// TIA Portal V18 export
// export: Created 2026-06-08T16:32:19.8720491Z, ExportSetting WithDefaults, DisplayName Totally Integrated Automation Portal, DisplayVersion V18, DisplayName TIA Portal Openness, DisplayVersion V18, DisplayName TIA Portal Version Control Interface, DisplayVersion V18, DisplayName STEP 7 Professional, DisplayVersion V18, DisplayName STEP 7 Safety, DisplayVersion V18, DisplayName WinCC Professional, DisplayVersion V18
VAR_GLOBAL   // PLC tag table "Default tag table"
   MachineCenter1_lid_start AT %Q3.5 : Bool;
   MachineCenter1_lid_produceLids AT %Q3.6 : Bool;
   push_excess_blue_base AT %Q3.7 : Bool;
   push_excess_green_base AT %Q4.0 : Bool;
   base_COUNTER_RESET_BUTTON_BLUE AT %I6.3 : Bool;
   base_COUNTER_RESET_BUTTON_GREEN AT %I6.4 : Bool;
   base_raw_excess_blue AT %Q4.1 : Bool;
   base_raw_excess_green AT %Q4.2 : Bool;
   base_vision_raw_execess_sensor_green AT %I6.5 : Bool;
   base_vision_raw_execess_sensor_blue AT %I6.6 : Bool;
   MachineCenter2_base_start AT %Q4.3 : Bool;
   Stop_blade4 AT %Q4.4 : Bool;
   Stop_blade5 AT %Q4.5 : Bool;
   MACHINE1_BUSY AT %I6.7 : Bool;
   BEGIN_SORTING_STATION_BASE_SENSOR AT %I7.0 : Bool;
   BEGIN_SORTING_STATION_BASE_1 AT %Q4.6 : Bool;
   BEGIN_SORTING_STATION_BASE_2 AT %Q4.7 : Bool;
   BEGIN_SORTING_STATION_BASE_3 AT %Q5.0 : Bool;
   Green_base_sorting_vision AT %I7.1 : Bool;
   Blue_base_sorting_vision AT %I7.2 : Bool;
   "Pusher_green_base (Front Limit)" AT %I7.3 : Bool;
   "Pusher_green_base (Back Limit)" AT %I7.4 : Bool;
   "Pusher_blue_base (Front Limit)" AT %I7.5 : Bool;
   "Pusher_blue_base (Back Limit)" AT %I7.6 : Bool;
   Pusher_blue_base_sorter AT %Q5.2 : Bool;
   Pusher_green_base_sorter AT %Q5.1 : Bool;
   Conv_sorting_set_lid AT %M2.7 : Bool;
   Emit_set_lid AT %M3.0 : Bool;
   Emit_set_base AT %M3.1 : Bool;
   "Blue count" AT %MW4 : Int;
   "excess blue lid raw led light" AT %Q5.4 : Bool;
   "excess green lid raw led light" AT %Q5.5 : Bool;
   "excess blue base raw led light" AT %Q5.6 : Bool;
   "excess green base raw led light" AT %Q5.7 : Bool;
   "blue lid sorting light" AT %Q6.0 : Bool;
   "green lid sorting light" AT %Q6.1 : Bool;
   "blue base sorting light" AT %Q6.2 : Bool;
   "green base sorting light" AT %Q6.3 : Bool;
   Green_Lid_conv_timer AT %T6 : Timer;
   Blue_Lid_conv_timer AT %T7 : Timer;
   Green_Base_conv_timer AT %T8 : Timer;
   Blue_Base_conv_timer AT %T9 : Timer;
END_VAR
